// Mitsubishi GX Works2 project: ZhaoQing_HuaCheng1_12_5_12_52   PLC: Q03UDE

TYPE ConveyorIO : STRUCT
  xCWPresent : BOOL;  (* 正转检测有无传感器 *)
  xCCWPresent : BOOL;  (* 反转检测有无传感器 *)
  xLoad : BOOL;  (* 上料请求 *)
  xUnload : BOOL;  (* 下料请求 *)
  xMotorCW : BOOL;  (* 电机正转 *)
  xMotorCCW : BOOL;  (* 电机反转 *)
  xEmpty : BOOL;  (* 线体状态为空 *)
  xNextRun : BOOL;  (* 下段线体运行 *)
  xLastRun : BOOL;  (* 上段线体运行 *)
  xUnloadCCW : BOOL;  (* 下料为反转 *)
  xloadCCW : BOOL;  (* 上料为反转 *)
  xLeave : BOOL;  (* 已经离开 *)
  xAuto : BOOL;  (* 自动 *)
  xManual : BOOL;  (* 手动 *)
  xForward : BOOL;  (* 正转手动 *)
  xBackward : BOOL;  (* 反转手动 *)
  strProductSerial : STRING[4];  (* 产品信息 *)
  xEStop : BOOL;  (* 急停 *)
  xReset : BOOL;  (* 复位 *)
  iProductCategory : INT;  (* 产品类型0：无料1：正极  2：负极 3：隔膜 4：空料架 *)
  xBusy : BOOL;  (* 工作中 *)
  tLeaveDelay : TIME;  (* 离开延时设置 *)
  xPutInto : BOOL;  (* 线体直接投入物料 *)
  xLoadAlarrm : BOOL;  (* 上料报警 *)
  xUnloadAlarm : BOOL;  (* 下料报警 *)
END_STRUCT END_TYPE

TYPE ShuttleCarIO : STRUCT
  xAuto : BOOL;  (* 自动 *)
  xManual : BOOL;  (* 手动 *)
  xReady : BOOL;  (* 准备就绪 *)
  xForward : BOOL;  (* 正转 *)
  xBackward : BOOL;  (* 反转 *)
  diCurrentPos : DINT;  (* 当前位置 *)
  diDestinationPos : DINT;  (* 目标位置 *)
  xCW : BOOL;  (* 正转输出 *)
  xCCW : BOOL;  (* 反转输出 *)
  xBrake : BOOL;  (* 刹车 *)
  xHomeSwitch : BOOL;  (* 零位接近开关 *)
  xPosLimit : BOOL;  (* 正限位 *)
  xNegLimit : BOOL;  (* 负限位 *)
  xMDIExe : BOOL;  (* MDI开始 *)
  xMDIDone : BOOL;  (* MDI 完成 *)
  xPassLimit : BOOL;  (* 限位屏蔽 *)
  xPosLimitCatch : BOOL;  (* 正限位捕捉 *)
  xNegLimitCatch : BOOL;  (* 负限位捕捉 *)
  xHomeExe : BOOL;  (* 开始寻零 *)
  xHomeDone : BOOL;  (* 寻零完成 *)
  xHomeBusy : BOOL;  (* 寻零中 *)
  xHomeFailed : BOOL;  (* 寻零失败 *)
  xBusy : BOOL;  (* 工作中 *)
  xReset : BOOL;  (* 复位 *)
  xEStop : BOOL;  (* 急停 *)
END_STRUCT END_TYPE

TYPE SwitchIO : STRUCT
  xAuto : BOOL;
  xManual : BOOL;
  xEStop : BOOL;
  xReset : BOOL;
  xLiftCylinderRetractDetect : BOOL;
  xLiftCylinderExtendDetect : BOOL;
  xLiftCylinderRetract : BOOL;
  xLiftCylinderExtend : BOOL;
  xEntryBarCylinderRetract : BOOL;
  xLiftCylinderExtendInit : BOOL;
  xEntryEnable : BOOL;
  xExitEnable : BOOL;
  xExitBarCylinderRetract : BOOL;
  xSwithEnable : BOOL;
  xLiftCylinderRetractButton : BOOL;
  xLiftCylinderExtendButton : BOOL;
  xEntryBarCylinderRetractButton : BOOL;
  xExitBarCylinderRetractButton : BOOL;
END_STRUCT END_TYPE

// global labels: Global1
VAR_GLOBAL
  g_xAuto : BOOL;
  g_xManual : BOOL;
  g_xEStop AT X23 : BOOL;
  g_xReset AT X20 : BOOL;
  g_xStackLampRed AT Y120 : BOOL;
  g_xStackLampAmber AT Y121 : BOOL;
  g_xStackLampGreen AT Y122 : BOOL;
  g_xBuzzer AT Y123 : BOOL;
  g_xStop AT M2 : BOOL;
  g_xLocalAutoStart AT M1 : BOOL;
  g_xRemoteAutoStart AT M0 : BOOL;
  g_xRemoteAuto AT M10 : BOOL;
  g_iState AT D40 : INT;
  g_iLocalAutoStep : INT;
END_VAR

// task Task_01 (event TRUE, interval 0, priority 31): POU, Start, UDP

PROGRAM POU
VAR
  H3000Conveyor1 : Conveyor;
  H3000Conveyor1IO : ConveyorIO;
  H3000Conveyor2 : Conveyor;
  H3000Conveyor2IO : ConveyorIO;
  H3000Conveyor3 : Conveyor;
  H3000Conveyor3IO : ConveyorIO;
  H3000Conveyor4 : Conveyor;
  H3000Conveyor4IO : ConveyorIO;
  H3000Conveyor5 : Conveyor;
  H3000Conveyor5IO : ConveyorIO;
  H3000Conveyor6 : Conveyor;
  H3000Conveyor6IO : ConveyorIO;
  H3000Conveyor7 : Conveyor;
  H3000Conveyor7IO : ConveyorIO;
  H3000Conveyor8 : Conveyor;
  H3000Conveyor8IO : ConveyorIO;
  H3000Conveyor9 : Conveyor;
  H3000Conveyor9IO : ConveyorIO;
  H3000Conveyor10 : Conveyor;
  H3000Conveyor10IO : ConveyorIO;
  H3000ChemConveyor1 : Conveyor;
  H3000ChemConveyor1IO : ConveyorIO;
  H3000ChemConveyor2 : Conveyor;
  H3000ChemConveyor2IO : ConveyorIO;
  H3000ChemConveyor3 : Conveyor;
  H3000ChemConveyor3IO : ConveyorIO;
  Lifter1 : ShuttleCar;
  Lifter1IO : ShuttleCarIO;
  Conveyor1 : Conveyor;
  Conveyor1IO : ConveyorIO;
  Lifter2 : ShuttleCar;
  Lifter2IO : ShuttleCarIO;
  Conveyor2 : Conveyor;
  Conveyor2IO : ConveyorIO;
  H2200Conveyor1 : Conveyor;
  H2200Conveyor1IO : ConveyorIO;
  H2200Conveyor2 : Conveyor;
  H2200Conveyor2IO : ConveyorIO;
  H2200Conveyor3 : Conveyor;
  H2200Conveyor3IO : ConveyorIO;
  H2200Conveyor4 : Conveyor;
  H2200Conveyor4IO : ConveyorIO;
  H2200Conveyor5 : Conveyor;
  H2200Conveyor5IO : ConveyorIO;
  H2200Conveyor6 : Conveyor;
  H2200Conveyor6IO : ConveyorIO;
  H2200Conveyor7 : Conveyor;
  H2200Conveyor7IO : ConveyorIO;
  H2200Conveyor8 : Conveyor;
  H2200Conveyor8IO : ConveyorIO;
  H2200Conveyor9 : Conveyor;
  H2200Conveyor9IO : ConveyorIO;
  H2200Conveyor10 : Conveyor;
  H2200Conveyor10IO : ConveyorIO;
  H1000Conveyor1 : Conveyor;
  H1000Conveyor1IO : ConveyorIO;
  H1000Conveyor2 : Conveyor;
  H1000Conveyor2IO : ConveyorIO;
  H1000Conveyor3 : Conveyor;
  H1000Conveyor3IO : ConveyorIO;
  H1000Conveyor4 : Conveyor;
  H1000Conveyor4IO : ConveyorIO;
  H1000Conveyor5 : Conveyor;
  H1000Conveyor5IO : ConveyorIO;
  H1000Conveyor6 : Conveyor;
  H1000Conveyor6IO : ConveyorIO;
  H1000Conveyor7 : Conveyor;
  H1000Conveyor7IO : ConveyorIO;
  H1000Conveyor8 : Conveyor;
  H1000Conveyor8IO : ConveyorIO;
  H1000Conveyor9 : Conveyor;
  H1000Conveyor9IO : ConveyorIO;
  H3000SwitchQuadPackage : Switch;
  H3000SwitchQuadPackageIO : SwitchIO;
  H3000SwitchChem : Switch;
  H3000SwitchChemIO : SwitchIO;
  H3000SwitchPackageConveyorIn : ConveyorIO;
  H3000SwitchPackageConveyorOut : ConveyorIO;
  H850Switch : Switch;
  H850SwitchIO : SwitchIO;
  H850SwitchConveyorIn : ConveyorIO;
  H850SwitchConveyorOut : ConveyorIO;
  H850Conveyor8 : Conveyor;
  H850Conveyor8IO : ConveyorIO;
  H1000Conveyor10 : Conveyor;
  H1000Conveyor10IO : ConveyorIO;
  H3000SwitchChemConveyorIn : ConveyorIO;
  H3000SwitchChemConveyorOut : ConveyorIO;
END_VAR
H3000SwitchQuadPackage(ConveyorEntryIO:=H3000SwitchPackageConveyorIn ,
                                                        ConveyorExitIO:=H3000SwitchPackageConveyorOut ,
                                                        SwitchIO:=H3000SwitchQuadPackageIO );
H3000SwitchQuadPackageIO.xAuto:=g_xAuto;
H3000SwitchQuadPackageIO.xManual:=g_xManual;
H3000SwitchQuadPackageIO.xReset:=g_xReset;
H3000SwitchQuadPackageIO.xLiftCylinderExtendButton:=M75;
H3000SwitchQuadPackageIO.xLiftCylinderRetractButton:=M76;
H3000SwitchQuadPackageIO.xExitBarCylinderRetractButton:=M83;
Y128:=H3000SwitchQuadPackageIO.xEXITBarCylinderRetract;
Y12C:=H3000SwitchQuadPackageIO.xLiftCylinderExtend;
Y12A:=H3000SwitchQuadPackageIO.xLiftCylinderRetract;
H3000SwitchQuadPackageIO.xLiftCylinderExtendDetect:=X29;
H3000SwitchQuadPackageIO.xLiftCylinderRetractDetect:=X2A;
H3000SwitchPackageConveyorIn.xForward:=M77;
H3000SwitchPackageConveyorIn.xCWPresent:=X28;
Y187:=H3000SwitchPackageConveyorIn.xMotorCW;
H3000SwitchPackageConveyorOut.xForward:=M78;
H3000SwitchPackageConveyorOut.xCWPresent:=X2B;
Y12B:=H3000SwitchPackageConveyorOut.xMotorCW;

H3000SwitchChem(ConveyorEntryIO:=H3000SwitchChemConveyorIn ,
                                                        ConveyorExitIO:=H3000SwitchChemConveyorOut ,
                                                        SwitchIO:=H3000SwitchChemIO );
H3000SwitchChemIO.xAuto:=g_xAuto;
H3000SwitchChemIO.xManual:=g_xManual;
H3000SwitchChemIO.xReset:=g_xReset;
H3000SwitchChemIO.xLiftCylinderExtendButton:=M79;
H3000SwitchChemIO.xLiftCylinderRetractButton:=M80;
Y129:=H3000SwitchChemIO.xLiftCylinderExtend;
Y12D:=H3000SwitchChemIO.xLiftCylinderRetract;
H3000SwitchChemIO.xLiftCylinderExtendDetect:=X2C;
H3000SwitchChemIO.xLiftCylinderRetractDetect:=X2D;
H3000SwitchChemConveyorIn.xForward:=M81;
H3000SwitchChemConveyorIn.xCWPresent:=X2E;
(*Y19B:=H3000SwitchPackageConveyorIn.xMotorCW;*)
H3000SwitchChemConveyorOut.xForward:=M82;
H3000SwitchChemConveyorOut.xCWPresent:=X2E;
Y12E:=H3000SwitchChemConveyorOut.xMotorCW;
H3000SwitchChemIO.xSwithEnable:=1;

Lifter1(ShuttleCarInOut:=Lifter1IO);
ShuttleCarCurrentPosition( X8C OR X8D ,X8C ,X8D, FALSE, Lifter1IO.diCurrentPos );
Lifter1IO.xAuto:=g_xAuto;
Lifter1IO.xManual:=g_xManual;
Lifter1IO.xEStop:=g_xEStop;
Lifter1IO.xReset:=g_xReset;
Lifter1IO.xReady:=X24;
Lifter1Io.xForward:=M50 OR X91;
Lifter1IO.xBackward:=M51 OR X92;
Lifter1IO.xPosLimit:=X8E;
Lifter1IO.xNegLimit:=X8F;
Y18D:=Lifter1IO.xCW;
Y18E:=Lifter1IO.xCCW;
Y192:=Lifter1IO.xBrake;

Conveyor1(ConveyorMotor:=Conveyor1IO);
Conveyor1IO.xAuto:=g_xAuto;
Conveyor1IO.xManual:=g_xManual;
Conveyor1IO.xReset:=g_xReset;
Conveyor1IO.tLeaveDelay:=T#2s;
Conveyor1IO.xForward:=M52;
Conveyor1IO.xBackward:=M53;
Conveyor1IO.xCWPresent:=X193;
Conveyor1IO.xCCWPresent:=X194;
Y18B:=Conveyor1IO.xMotorCW;
Y18C:=Conveyor1IO.xMotorCCW;

Lifter2(ShuttleCarInOut:=Lifter2IO);
ShuttleCarCurrentPosition( X96 OR X97 ,X96 ,X97, FALSE, Lifter2IO.diCurrentPos );
Lifter2IO.xAuto:=g_xAuto;
Lifter2IO.xManual:=g_xManual;
Lifter2IO.xEStop:=g_xEStop;
Lifter2IO.xReset:=g_xReset;
Lifter2IO.xReady:=X25;
Lifter2Io.xForward:=M54 OR X9B;
Lifter2IO.xBackward:=M55 OR X9C;
Lifter2IO.xPosLimit:=X98;
Lifter2IO.xNegLimit:=X99;
Y193:=Lifter2IO.xCW;
Y194:=Lifter2IO.xCCW;
Y198:=Lifter2IO.xBrake;

Conveyor2(ConveyorMotor:=Conveyor2IO);
Conveyor2IO.xAuto:=g_xAuto;
Conveyor2IO.xManual:=g_xManual;
Conveyor2IO.xReset:=g_xReset;
Conveyor2IO.tLeaveDelay:=T#2s;
Conveyor2IO.xForward:=M56;
Conveyor2IO.xBackward:=M57;
Conveyor2IO.xCWPresent:=X93;
Conveyor2IO.xCCWPresent:=X94;
Y199:=Conveyor2IO.xMotorCW;
Y19A:=Conveyor2IO.xMotorCCW;


H3000Conveyor1(ConveyorMotor:=H3000Conveyor1IO);
H3000Conveyor1IO.xAuto:=g_xAuto;
H3000Conveyor1IO.xManual:=g_xManual;
H3000Conveyor1IO.xReset:=g_xReset;
H3000Conveyor1IO.tLeaveDelay:=t#2s;
H3000Conveyor1IO.xForward:=M30;
H3000Conveyor1IO.xCWPresent:=X2F;
Y12F:=H3000Conveyor1IO.xMotorCW;

H3000Conveyor2(ConveyorMotor:=H3000Conveyor2IO);
H3000Conveyor2IO.xAuto:=g_xAuto;
H3000Conveyor2IO.xManual:=g_xManual;
H3000Conveyor2IO.xReset:=g_xReset;
H3000Conveyor2IO.tLeaveDelay:=t#2s;
H3000Conveyor2IO.xForward:=M31;
H3000Conveyor2IO.xCWPresent:=X30;
Y130:=H3000Conveyor2IO.xMotorCW;

H3000Conveyor3(ConveyorMotor:=H3000Conveyor3IO);
H3000Conveyor3IO.xAuto:=g_xAuto;
H3000Conveyor3IO.xManual:=g_xManual;
H3000Conveyor3IO.xReset:=g_xReset;
H3000Conveyor3IO.tLeaveDelay:=t#2s;
H3000Conveyor3IO.xForward:=M32;
H3000Conveyor3IO.xCWPresent:=X31;
Y131:=H3000Conveyor3IO.xMotorCW;

H3000Conveyor4(ConveyorMotor:=H3000Conveyor4IO);
H3000Conveyor4IO.xAuto:=g_xAuto;
H3000Conveyor4IO.xManual:=g_xManual;
H3000Conveyor4IO.xReset:=g_xReset;
H3000Conveyor4IO.tLeaveDelay:=t#2s;
H3000Conveyor4IO.xForward:=M33;
H3000Conveyor4IO.xCWPresent:=X32;
Y132:=H3000Conveyor4IO.xMotorCW;

H3000Conveyor5(ConveyorMotor:=H3000Conveyor5IO);
H3000Conveyor5IO.xAuto:=g_xAuto;
H3000Conveyor5IO.xManual:=g_xManual;
H3000Conveyor5IO.xReset:=g_xReset;
H3000Conveyor5IO.tLeaveDelay:=t#2s;
H3000Conveyor5IO.xForward:=M34;
H3000Conveyor5IO.xCWPresent:=X33;
Y133:=H3000Conveyor5IO.xMotorCW;

H3000Conveyor6(ConveyorMotor:=H3000Conveyor6IO);
H3000Conveyor6IO.xAuto:=g_xAuto;
H3000Conveyor6IO.xManual:=g_xManual;
H3000Conveyor6IO.xReset:=g_xReset;
H3000Conveyor6IO.tLeaveDelay:=t#2s;
H3000Conveyor6IO.xForward:=M34;
H3000Conveyor6IO.xCWPresent:=X34;
Y134:=H3000Conveyor6IO.xMotorCW;

H3000Conveyor7(ConveyorMotor:=H3000Conveyor7IO);
H3000Conveyor7IO.xAuto:=g_xAuto;
H3000Conveyor7IO.xManual:=g_xManual;
H3000Conveyor7IO.xReset:=g_xReset;
H3000Conveyor7IO.tLeaveDelay:=t#2s;
H3000Conveyor7IO.xForward:=M35;
H3000Conveyor7IO.xCWPresent:=X35;
Y135:=H3000Conveyor7IO.xMotorCW;

H3000Conveyor8(ConveyorMotor:=H3000Conveyor8IO);
H3000Conveyor8IO.xAuto:=g_xAuto;
H3000Conveyor8IO.xManual:=g_xManual;
H3000Conveyor8IO.xReset:=g_xReset;
H3000Conveyor8IO.tLeaveDelay:=t#2s;
H3000Conveyor8IO.xForward:=M36;
H3000Conveyor8IO.xCWPresent:=X36;
Y136:=H3000Conveyor8IO.xMotorCW;

H3000Conveyor9(ConveyorMotor:=H3000Conveyor9IO);
H3000Conveyor9IO.xAuto:=g_xAuto;
H3000Conveyor9IO.xManual:=g_xManual;
H3000Conveyor9IO.xReset:=g_xReset;
H3000Conveyor9IO.tLeaveDelay:=t#2s;
H3000Conveyor9IO.xForward:=M37;
H3000Conveyor9IO.xCWPresent:=X37;
Y137:=H3000Conveyor9IO.xMotorCW;

H3000Conveyor10(ConveyorMotor:=H3000Conveyor10IO);
H3000Conveyor10IO.xAuto:=g_xAuto;
H3000Conveyor10IO.xManual:=g_xManual;
H3000Conveyor10IO.xReset:=g_xReset;
H3000Conveyor10IO.tLeaveDelay:=t#2s;
H3000Conveyor10IO.xForward:=M38;
H3000Conveyor10IO.xCWPresent:=X38;
Y138:=H3000Conveyor10IO.xMotorCW;

H3000ChemConveyor1(ConveyorMotor:=H3000ChemConveyor1IO);
H3000ChemConveyor1IO.xAuto:=g_xAuto;
H3000ChemConveyor1IO.xManual:=g_xManual;
H3000ChemConveyor1IO.xReset:=g_xReset;
H3000ChemConveyor1IO.tLeaveDelay:=t#2s;
H3000ChemConveyor1IO.xForward:=M39;
H3000ChemConveyor1IO.xCWPresent:=X39;
Y139:=H3000ChemConveyor1IO.xMotorCW;

H3000ChemConveyor2(ConveyorMotor:=H3000ChemConveyor2IO);
H3000ChemConveyor2IO.xAuto:=g_xAuto;
H3000ChemConveyor2IO.xManual:=g_xManual;
H3000ChemConveyor2IO.xReset:=g_xReset;
H3000ChemConveyor2IO.tLeaveDelay:=t#2s;
H3000ChemConveyor2IO.xForward:=M40;
H3000ChemConveyor2IO.xCWPresent:=X3A;
Y13A:=H3000ChemConveyor2IO.xMotorCW;

H3000ChemConveyor3(ConveyorMotor:=H3000ChemConveyor3IO);
H3000ChemConveyor3IO.xAuto:=g_xAuto;
H3000ChemConveyor3IO.xManual:=g_xManual;
H3000ChemConveyor3IO.xReset:=g_xReset;
H3000ChemConveyor3IO.tLeaveDelay:=t#2s;
H3000ChemConveyor3IO.xForward:=M41;
H3000ChemConveyor3IO.xCWPresent:=X3B;
Y13B:=H3000ChemConveyor3IO.xMotorCW;

H2200Conveyor1(ConveyorMotor:=H2200Conveyor1IO);
H2200Conveyor1IO.xAuto:=g_xAuto;
H2200Conveyor1IO.xManual:=g_xManual;
H2200Conveyor1IO.xReset:=g_xReset;
H2200Conveyor1IO.tLeaveDelay:=t#2s;
H2200Conveyor1IO.xForward:=M42;
H2200Conveyor1IO.xCWPresent:=X3F;
Y13F:=H2200Conveyor1IO.xMotorCW;

H2200Conveyor2(ConveyorMotor:=H2200Conveyor2IO);
H2200Conveyor2IO.xAuto:=g_xAuto;
H2200Conveyor2IO.xManual:=g_xManual;
H2200Conveyor2IO.xReset:=g_xReset;
H2200Conveyor2IO.tLeaveDelay:=t#2s;
H2200Conveyor2IO.xForward:=M43;
H2200Conveyor2IO.xCWPresent:=X40;
Y140:=H2200Conveyor2IO.xMotorCW;

H2200Conveyor3(ConveyorMotor:=H2200Conveyor3IO);
H2200Conveyor3IO.xAuto:=g_xAuto;
H2200Conveyor3IO.xManual:=g_xManual;
H2200Conveyor3IO.xReset:=g_xReset;
H2200Conveyor3IO.tLeaveDelay:=t#2s;
H2200Conveyor3IO.xForward:=M44;
H2200Conveyor3IO.xCWPresent:=X41;
Y141:=H2200Conveyor2IO.xMotorCW;

H2200Conveyor4(ConveyorMotor:=H2200Conveyor4IO);
H2200Conveyor4IO.xAuto:=g_xAuto;
H2200Conveyor4IO.xManual:=g_xManual;
H2200Conveyor4IO.xReset:=g_xReset;
H2200Conveyor4IO.tLeaveDelay:=t#2s;
H2200Conveyor4IO.xForward:=M45;
H2200Conveyor4IO.xCWPresent:=X42;
Y142:=H2200Conveyor2IO.xMotorCW;

H2200Conveyor5(ConveyorMotor:=H2200Conveyor5IO);
H2200Conveyor5IO.xAuto:=g_xAuto;
H2200Conveyor5IO.xManual:=g_xManual;
H2200Conveyor5IO.xReset:=g_xReset;
H2200Conveyor5IO.tLeaveDelay:=t#2s;
H2200Conveyor5IO.xForward:=M46;
H2200Conveyor5IO.xCWPresent:=X43;
Y143:=H2200Conveyor2IO.xMotorCW;

H2200Conveyor6(ConveyorMotor:=H2200Conveyor6IO);
H2200Conveyor6IO.xAuto:=g_xAuto;
H2200Conveyor6IO.xManual:=g_xManual;
H2200Conveyor6IO.xReset:=g_xReset;
H2200Conveyor6IO.tLeaveDelay:=t#2s;
H2200Conveyor6IO.xForward:=M47;
H2200Conveyor6IO.xCWPresent:=X44;
Y144:=H2200Conveyor6IO.xMotorCW;

H2200Conveyor7(ConveyorMotor:=H2200Conveyor7IO);
H2200Conveyor7IO.xAuto:=g_xAuto;
H2200Conveyor7IO.xManual:=g_xManual;
H2200Conveyor7IO.xReset:=g_xReset;
H2200Conveyor7IO.tLeaveDelay:=t#2s;
H2200Conveyor7IO.xForward:=M48;
H2200Conveyor7IO.xCWPresent:=X45;
Y145:=H2200Conveyor7IO.xMotorCW;

H2200Conveyor8(ConveyorMotor:=H2200Conveyor8IO);
H2200Conveyor8IO.xAuto:=g_xAuto;
H2200Conveyor8IO.xManual:=g_xManual;
H2200Conveyor8IO.xReset:=g_xReset;
H2200Conveyor8IO.tLeaveDelay:=t#2s;
H2200Conveyor8IO.xForward:=M49;
H2200Conveyor8IO.xCWPresent:=X46;
Y146:=H2200Conveyor8IO.xMotorCW;

H2200Conveyor9(ConveyorMotor:=H2200Conveyor9IO);
H2200Conveyor9IO.xAuto:=g_xAuto;
H2200Conveyor9IO.xManual:=g_xManual;
H2200Conveyor9IO.xReset:=g_xReset;
H2200Conveyor9IO.tLeaveDelay:=t#2s;
H2200Conveyor9IO.xForward:=M58;
H2200Conveyor9IO.xCWPresent:=X47;
Y147:=H2200Conveyor9IO.xMotorCW;

H2200Conveyor10(ConveyorMotor:=H2200Conveyor10IO);
H2200Conveyor10IO.xAuto:=g_xAuto;
H2200Conveyor10IO.xManual:=g_xManual;
H2200Conveyor10IO.xReset:=g_xReset;
H2200Conveyor10IO.tLeaveDelay:=t#2s;
H2200Conveyor10IO.xForward:=M59;
H2200Conveyor10IO.xCWPresent:=X48;
Y148:=H2200Conveyor10IO.xMotorCW;

H1000Conveyor1(ConveyorMotor:=H1000Conveyor1IO);
H1000Conveyor1IO.xAuto:=g_xAuto;
H1000Conveyor1IO.xManual:=g_xManual;
H1000Conveyor1IO.xReset:=g_xReset;
H1000Conveyor1IO.tLeaveDelay:=t#2s;
H1000Conveyor1IO.xForward:=M60;
H1000Conveyor1IO.xCWPresent:=X49;
Y149:=H1000Conveyor1IO.xMotorCW;

H1000Conveyor2(ConveyorMotor:=H1000Conveyor2IO);
H1000Conveyor2IO.xAuto:=g_xAuto;
H1000Conveyor2IO.xManual:=g_xManual;
H1000Conveyor2IO.xReset:=g_xReset;
H1000Conveyor2IO.tLeaveDelay:=t#2s;
H1000Conveyor2IO.xForward:=M61;
H1000Conveyor2IO.xCWPresent:=X4A;
Y14A:=H1000Conveyor2IO.xMotorCW;

H1000Conveyor3(ConveyorMotor:=H1000Conveyor3IO);
H1000Conveyor3IO.xAuto:=g_xAuto;
H1000Conveyor3IO.xManual:=g_xManual;
H1000Conveyor3IO.xReset:=g_xReset;
H1000Conveyor3IO.tLeaveDelay:=t#2s;
H1000Conveyor3IO.xForward:=M62;
H1000Conveyor3IO.xCWPresent:=X4B;
Y14B:=H1000Conveyor3IO.xMotorCW;

H1000Conveyor4(ConveyorMotor:=H1000Conveyor4IO);
H1000Conveyor4IO.xAuto:=g_xAuto;
H1000Conveyor4IO.xManual:=g_xManual;
H1000Conveyor4IO.xReset:=g_xReset;
H1000Conveyor4IO.tLeaveDelay:=t#2s;
H1000Conveyor4IO.xForward:=M63;
H1000Conveyor4IO.xCWPresent:=X4C;
Y14C:=H1000Conveyor4IO.xMotorCW;

H1000Conveyor5(ConveyorMotor:=H1000Conveyor5IO);
H1000Conveyor5IO.xAuto:=g_xAuto;
H1000Conveyor5IO.xManual:=g_xManual;
H1000Conveyor5IO.xReset:=g_xReset;
H1000Conveyor5IO.tLeaveDelay:=t#2s;
H1000Conveyor5IO.xForward:=M64;
H1000Conveyor5IO.xCWPresent:=X4D;
Y14D:=H1000Conveyor1IO.xMotorCW;

H1000Conveyor6(ConveyorMotor:=H1000Conveyor6IO);
H1000Conveyor6IO.xAuto:=g_xAuto;
H1000Conveyor6IO.xManual:=g_xManual;
H1000Conveyor6IO.xReset:=g_xReset;
H1000Conveyor6IO.tLeaveDelay:=t#2s;
H1000Conveyor6IO.xForward:=M65;
H1000Conveyor6IO.xCWPresent:=X4E;
Y14E:=H1000Conveyor1IO.xMotorCW;

H1000Conveyor7(ConveyorMotor:=H1000Conveyor7IO);
H1000Conveyor7IO.xAuto:=g_xAuto;
H1000Conveyor7IO.xManual:=g_xManual;
H1000Conveyor7IO.xReset:=g_xReset;
H1000Conveyor7IO.tLeaveDelay:=t#2s;
H1000Conveyor7IO.xForward:=M66;
H1000Conveyor7IO.xCWPresent:=X4F;
Y14F:=H1000Conveyor1IO.xMotorCW;

H1000Conveyor8(ConveyorMotor:=H1000Conveyor8IO);
H1000Conveyor8IO.xAuto:=g_xAuto;
H1000Conveyor8IO.xManual:=g_xManual;
H1000Conveyor8IO.xReset:=g_xReset;
H1000Conveyor8IO.tLeaveDelay:=t#2s;
H1000Conveyor8IO.xForward:=M67;
H1000Conveyor8IO.xCWPresent:=X50;
Y150:=H1000Conveyor8IO.xMotorCW;

H850Switch(ConveyorEntryIO:=H850SwitchConveyorIn,ConveyorExitIO:=H850SwitchConveyorOut,SwitchIO:=H850SwitchIO);
H850SwitchIO.xAuto:=g_xAuto;
H850SwitchIO.xManual:=g_xManual;
H850SwitchIO.xReset:=g_xReset;
H850SwitchIO.xLiftCylinderExtendButton:=M71;
H850SwitchIO.xLiftCylinderRetractButton:=M72;
Y189:=H850SwitchIO.xLiftCylinderExtend;
Y188:=H850SwitchIO.xLiftCylinderRetract;
H850SwitchIO.xLiftCylinderExtendDetect:=X88;
H850SwitchIO.xLiftCylinderRetractDetect:=X89;
H850SwitchConveyorIn.xForward:=M70;
H850SwitchConveyorIn.xCWPresent:=XB4;
Y19B:=H850SwitchConveyorIn.xMotorCW;
H850SwitchConveyorOut.xForward:=M73;
H850SwitchConveyorOut.xCWPresent:=X8A;
Y18A:=H850SwitchConveyorOut.xMotorCW;


H850Conveyor8(ConveyorMotor:=H850Conveyor8IO);
H850Conveyor8IO.xAuto:=g_xAuto;
H850Conveyor8IO.xManual:=g_xManual;
H850Conveyor8IO.xReset:=g_xReset;
H850Conveyor8IO.tLeaveDelay:=t#2s;
H850Conveyor8IO.xForward:=M74;
H850Conveyor8IO.xCWPresent:=X7F;
Y17F:=H850Conveyor8IO.xMotorCW;

IF g_xAuto THEN
	H3000SwitchQuadPackageIO.xEntryEnable:=M881;
	H3000SwitchQuadPackageIO.xSwithEnable:=1;
	H3000SwitchQuadPackageio.xExitEnable:=H3000Conveyor1IO.xEmpty;
	H3000Conveyor1Io.xLoad:=H3000SwitchPackageConveyorOut.xNextRun;
	H3000Conveyor1IO.xUnload:=H3000Conveyor2IO.xEmpty;
	H3000Conveyor2IO.xLoad:=H3000Conveyor1IO.xNextRun;
	H3000Conveyor2IO.xUnload:=H3000Conveyor3IO.xEmpty;
	H3000Conveyor3IO.xLoad:=H3000Conveyor2IO.xNextRun;	
	H3000Conveyor3IO.xUnload:=H3000Conveyor4IO.xEmpty;
	H3000Conveyor4IO.xLoad:=H3000Conveyor3IO.xNextRun;
	H3000Conveyor4IO.xUnload:=H3000Conveyor5IO.xEmpty;
	H3000Conveyor5IO.xLoad:=H3000Conveyor4IO.xNextRun;
	H3000Conveyor5IO.xUnload:=H3000Conveyor6IO.xEmpty;
	H3000Conveyor6IO.xLoad:=H3000Conveyor5IO.xNextRun;
	H3000Conveyor6IO.xUnload:=H3000Conveyor7IO.xEmpty;
	H3000Conveyor7IO.xLoad:=H3000Conveyor6IO.xNextRun;
	H3000Conveyor7IO.xUnload:=H3000Conveyor8IO.xEmpty;
	H3000Conveyor8IO.xLoad:=H3000Conveyor7IO.xNextRun;	
	H3000Conveyor8IO.xUnload:=H3000Conveyor9IO.xEmpty;
	H3000Conveyor9IO.xLoad:=H3000Conveyor8IO.xNextRun;	
	H3000Conveyor9IO.xUnload:=H3000Conveyor10IO.xEmpty;
	H3000Conveyor10IO.xLoad:=H3000Conveyor9IO.xNextRun;
	
	H2200Conveyor1IO.xLoad:=M201;
	H2200Conveyor1IO.xUnload:=H2200Conveyor2IO.xEmpty;
	H2200Conveyor2IO.xLoad:=H2200Conveyor1IO.xNextRun;
	H2200Conveyor2IO.xUnload:=H2200Conveyor3IO.xEmpty;
	H2200Conveyor3IO.xLoad:=H2200Conveyor2IO.xNextRun;	
	H2200Conveyor3IO.xUnload:=H2200Conveyor4IO.xEmpty;
	H2200Conveyor4IO.xLoad:=H2200Conveyor3IO.xNextRun;
	H2200Conveyor4IO.xUnload:=H2200Conveyor5IO.xEmpty;
	H2200Conveyor5IO.xLoad:=H2200Conveyor4IO.xNextRun;
	H2200Conveyor5IO.xUnload:=H2200Conveyor6IO.xEmpty;
	H2200Conveyor6IO.xLoad:=H2200Conveyor5IO.xNextRun;
	H2200Conveyor6IO.xUnload:=H2200Conveyor7IO.xEmpty;
	H2200Conveyor7IO.xLoad:=H2200Conveyor6IO.xNextRun;
	H2200Conveyor7IO.xUnload:=H2200Conveyor8IO.xEmpty;
	H2200Conveyor8IO.xLoad:=H2200Conveyor7IO.xNextRun;	
	H2200Conveyor8IO.xUnload:=H2200Conveyor9IO.xEmpty;
	H2200Conveyor9IO.xLoad:=H2200Conveyor8IO.xNextRun;	
	H2200Conveyor9IO.xUnload:=H2200Conveyor10IO.xEmpty;
	H2200Conveyor10IO.xLoad:=H2200Conveyor9IO.xNextRun;
	
	H1000Conveyor10IO.xLoad:=M202;
	H1000Conveyor10IO.xUnload:=H1000Conveyor9IO.xEmpty;
    H1000Conveyor9IO.xLoad:=H1000Conveyor10IO.xNextRun;
    H1000Conveyor9IO.xUnload:=H1000Conveyor8IO.xEmpty;
    H1000Conveyor8IO.xLoad:=H1000Conveyor9IO.xNextRun;
    H1000Conveyor8IO.xUnload:=H1000Conveyor7IO.xEmpty;
    H1000Conveyor7IO.xLoad:=H1000Conveyor8IO.xNextRun;
    H1000Conveyor7IO.xUnload:=H1000Conveyor6IO.xEmpty;
    H1000Conveyor6IO.xLoad:=H1000Conveyor7IO.xNextRun;
    H1000Conveyor6IO.xUnload:=H1000Conveyor5IO.xEmpty;
    H1000Conveyor5IO.xLoad:=H1000Conveyor6IO.xNextRun;
    H1000Conveyor5IO.xUnload:=H1000Conveyor4IO.xEmpty;
    H1000Conveyor4IO.xLoad:=H1000Conveyor5IO.xNextRun;
    H1000Conveyor4IO.xUnload:=H1000Conveyor3IO.xEmpty;
    H1000Conveyor3IO.xLoad:=H1000Conveyor4IO.xNextRun;
    H1000Conveyor3IO.xUnload:=H1000Conveyor2IO.xEmpty;
    H1000Conveyor2IO.xLoad:=H1000Conveyor3IO.xNextRun;  
    H1000Conveyor2IO.xUnload:=H1000Conveyor1IO.xEmpty;
    H1000Conveyor1IO.xLoad:=H1000Conveyor2IO.xNextRun;      
	
	H850SwitchIO.xEntryEnable:=M880;
	H850SwitchIO.xSwithEnable:=1;
	H850SwitchIO.xExitEnable:=H850Conveyor8IO.xEmpty;
    H850Conveyor8IO.xLoad:=H850SwitchConveyorOut.xNextRun;
    
    
    
END_IF;
END_PROGRAM

FUNCTION_BLOCK Conveyor
VAR
  tRundelay : TIME;  (* 离开延时 *)
END_VAR
VAR_IN_OUT
  ConveyorMotor : ConveyorIO;  (* 输送线输入输出 *)
END_VAR
VAR
  iStep : INT;  (* 上料步骤 *)
  m_tLoadTimer : TIME;  (* 上料计时器 *)
  m_tUnloadTimer : TIME;  (* 下料计时器 *)
  m_tonLeaveDelay : TON;  (* 离开延时定时器 *)
  m_xLeaveDelayOut : BOOL;  (* 离开延时 *)
  m_tLeaveCurrentTime : TIME;
  m_tonLoadAlarm : TON;  (* 上料延时报警 *)
END_VAR
VAR CONSTANT
  LOAD_UNLOAD_TIME : TIME := T#30s;  (* 延时报警常量 *)
END_VAR
VAR
  m_tonUnloadAlam : TON;  (* 下料报警定时器 *)
END_VAR
(*////////////////////////////////////////////////////////////////////////////////////////////////////////////
//传输线控制FB块，可控制单方向线体，双向旋转线体，支持双向上下料            
//线体初始化后为空的情况下输入xLoad信号即可进行上料动作，使用xLoadCCW信号可反方向上料
//增加了产品信息和产品种类的储存，当传输线为空和上料进行标志位为零的情况下清除产品信息和产品种类
//使用方式是在置位xLoad信号后，把产品信息和产品种类传入，等下料后自动清零
//线体不为空的情况下使用xUnload信号可进行下料动作，物料有无传感器的下降沿后出发计时器，延时断开传输线旋转
//单方向传输线体把xLoadCCW、xUnloadCCW设置为零，双向线体上料方向和下料反向的,方向固定的 把xUnloadCCW设置为1
//双方向线体双向都能上下料的要根据上料的方向来设置xLoadCCW,xUnloadCCW
//增加工作中信号xBusy当电机正转 显示为工作中
//增加上下料超时报警，xLoadAlarm，xUnloadAlarm，设定时间在LOAD_UNLOAD_TIME常量上，现在设置的为30秒
//增加xPutInto信号，用于直接投入的物料，检测开关感应到后，直接进入下料流程，上升沿有效
//离开延时改为变量 iLeaveDelay 默认为0 离开检测开关离输送线尾端比较远的线体需要根据情况设定100ms为单位
//修改信息  修改后请增加版本
//YAO      V1.0
///////////////////////////////////////////////////////////////////////////////////////////////////////////
********************************************************)


IF ConveyorMotor.xAuto THEN
CASE iStep OF
	0:
	ConveyorMotor.xMotorCW:=0;
	ConveyorMotor.xMotorCCW:=0;
	ConveyorMotor.xNextRun:=0;

	IF (ConveyorMotor.xCWPresent OR ConveyorMotor.xCCWPresent) 
		AND ConveyorMotor.xEStop=0 
		AND ConveyorMotor.xLoadAlarrm = 0
		AND ConveyorMotor.xUnloadAlarm = 0 THEN
		iStep:=3;
		ConveyorMotor.xEmpty:=0;
		ELSE
		iStep:=1;
		ConveyorMotor.xEmpty:=1;
	END_IF;
		
	1: 
	IF ConveyorMotor.xLoad    
		AND ConveyorMotor.xMotorCW=0   
		AND ConveyorMotor.xMotorCCW=0   
		AND ConveyorMotor.xEmpty THEN	
		iStep:=2;
	END_IF;
	2: 
	IF ConveyorMotor.xloadCCW THEN
		ConveyorMotor.xMotorCCW:=1; 
		ConveyorMotor.xMotorCW:=0;
		IF ConveyorMotor.xCCWPresent THEN
			iStep:=3;
		END_IF;
		ELSE
	    ConveyorMotor.xMotorCW:=1;  
		ConveyorMotor.xMotorCCW:=0;
	    IF ConveyorMotor.xCWPresent THEN 	 
		    iStep:=3;
		END_IF;
	END_IF;
	3:
	ConveyorMotor.xMotorCW:=0;
	ConveyorMotor.xMotorCCW:=0;
	ConveyorMotor.xEmpty:=0;
	IF ConveyorMotor.xUnload THEN 
		iStep:=4;
	END_IF;
	4:	
	IF ConveyorMotor.xUnloadCCW THEN   
		ConveyorMotor.xMotorCCW:=1;  
		ConveyorMotor.xMotorCW:=0;

		ConveyorMotor.xLeave:=ldf(TRUE,ConveyorMotor.xCCWPresent) OR ConveyorMotor.xLeave;
		ELSE
	    ConveyorMotor.xMotorCW:=1;  
		ConveyorMotor.xMotorCCW:=0;
		ConveyorMotor.xLeave:=ldf(TRUE,ConveyorMotor.xCWPresent) OR ConveyorMotor.xLeave;
	END_IF;
	ConveyorMotor.xNextRun:=1; 
	m_tonLeaveDelay(IN:= ConveyorMotor.xLeave,PT:= ConveyorMotor.tLeaveDelay,Q:=m_xLeaveDelayOut ,ET:= m_tLeaveCurrentTime );	
	IF m_xLeaveDelayOut THEN
		ConveyorMotor.xMotorCW:=0;
		ConveyorMotor.xMotorCCW:=0;
		iStep:=0;
		ConveyorMotor.xNextRun:=0;
		ConveyorMotor.xLeave:=0;
		ConveyorMotor.xEmpty:=1;		
	END_IF;	
	IF NOT ConveyorMotor.xUnload THEN 
		istep:=0;
	END_IF;
END_CASE;
IF LDP(TRUE,ConveyorMotor.xPutInto) THEN
	iStep:=0;
END_IF;
END_IF;
IF ConveyorMotor.xEmpty AND NOT ConveyorMotor.xLoad THEN
	ConveyorMotor.strProductSerial:='';
	ConveyorMotor.iProductCategory:=0;
END_IF;
IF ConveyorMotor.xEStop OR ConveyorMotor.xReset THEN
	iStep:=0;
END_IF;	

IF ConveyorMotor.xManual THEN
	iStep:=0;

	IF ConveyorMotor.xForward 
		AND ConveyorMotor.xBackward=0 
		AND ConveyorMotor.xMotorCCW=0 THEN
		ConveyorMotor.xMotorCW:=1;
		ConveyorMotor.xMotorCCW:=0;
		ELSE
		ConveyorMotor.xMotorCW:=0;
	END_IF;

	IF ConveyorMotor.xBackward 
		AND ConveyorMotor.xForward=0 
		AND ConveyorMotor.xMotorCW=0  THEN
		ConveyorMotor.xMotorCCW:=1;
		conveyormotor.xMotorCW:=0;
		ELSE
		ConveyorMotor.xMotorCCW:=0;
	END_IF;
END_IF;
IF ConveyorMotor.xMotorCCW        
	OR ConveyorMotor.xMotorCW THEN  
	ConveyorMotor.xBusy:=1;
	ELSE
	ConveyorMotor.xBusy:=0;
END_IF;
m_tonLoadAlarm(IN:= iStep=2 ,PT:= LOAD_UNLOAD_TIME,Q:= ConveyorMotor.xLoadAlarrm ,ET:= m_tLoadTimer );
m_tonUnloadAlam(IN:= iStep=4,PT:= LOAD_UNLOAD_TIME,Q:= ConveyorMotor.xUnloadAlarm,ET:= m_tUnloadTimer );
(*OUT_T(iStep=2,m_tLoadTimer,LOAD_UNLOAD_TIME);
OUT_T(iStep=4,m_tUnloadTimer,LOAD_UNLOAD_TIME);
ConveyorMotor.xLoadAlarrm:=m_tLoadTimer.S;
ConveyorMotor.xUnloadAlarm:=m_tUnloadTimer.S;*)
END_FUNCTION_BLOCK

FUNCTION_BLOCK ShuttleCar
VAR_IN_OUT
  ShuttleCarInOut : ShuttleCarIO;
END_VAR
VAR
  m_xBrakeDelay : BOOL;  (* 刹车延时标志位 *)
  diCurrentPosRetain : DINT;
  m_tonBrakeDelay : TON;  (* 延时 *)
  m_tBrakeDelay : TIME;
  m_xBrake : BOOL;
  m_tBrakeDelayCurrentTime : TIME;
END_VAR
(*******************************************************************
输送小车程序，可用于使用认址片控制位置的输送车程序，可用于控制提升机，
使用了限位捕捉程序防止小车惯性过大冲过限位后继续行走，捕捉程序采用反
转复位，这样设计有弊端可能反转复位后车的位置并没有回到限位以内,当两个
限位同时碰到的时候，会使运料小车进入死锁状态，通过xPassLimit来解开死锁，
可以在触摸屏中使用一个带权限的按钮来进行控制，配合ShuttleCarCurrentPos
函数来计算位置信息
修改信息  修改后请增加版本
YAO      V1.0
********************************************************************)

ShuttleCarInOut.xPosLimitCatch:=LDF(TRUE,ShuttleCarInOut.xPosLimit) OR ShuttleCarInOut.xPosLimitCatch;
IF ShuttleCarInOut.xCCW THEN  
	ShuttleCarInOut.xPosLimitCatch:=0;
END_IF;

ShuttleCarInOut.xNegLimitCatch:=LDF(TRUE,ShuttleCarInOut.xNegLimit) OR ShuttleCarInOut.xNegLimitCatch;
IF ShuttleCarInOut.xCW THEN   
	ShuttleCarInOut.xNegLimitCatch:=0;  
END_IF;
IF ShuttleCarInOut.xPassLimit OR
	(ShuttleCarInOut.xNegLimitCatch 
	AND ShuttleCarInOut.xPosLimitCatch)  THEN  
	ShuttleCarInOut.xNegLimitCatch:=0; 
	ShuttleCarInOut.xPosLimitCatch:=0;
END_IF;

IF ShuttleCarInOut.xReady THEN	
    IF ShuttleCarInOut.xManual THEN  
	    IF ShuttleCarInOut.xForward 
			AND ShuttleCarInOut.xBackward=0 
			AND ShuttleCarInOut.xCCW=0 
			AND ShuttleCarInOut.xPosLimitCatch=0 
			AND ShuttleCarInOut.xEStop THEN
		    ShuttleCarInOut.xCW:=1;
		    ELSE
		    ShuttleCarInOut.xCW:=0;
	    END_IF;
	    IF ShuttleCarInOut.xBackward 
			AND ShuttleCarInOut.xForward=0 
			AND ShuttleCarInOut.xCW=0 
			AND ShuttleCarInOut.xNegLimitCatch=0 
			AND ShuttleCarInOut.xEStop THEN  
		    ShuttleCarInOut.xCCW:=1;
		    ELSE
		    ShuttleCarInOut.xCCW:=0;
	    END_IF;
    END_IF;
  IF ShuttleCarInOut.xAuto AND ShuttleCarInOut.xEStop THEN  
	  IF ShuttleCarInOut.xMDIExe AND ShuttleCarInOut.diDestinationPos<>0 THEN
	
	    IF ShuttleCarInOut.diCurrentPos<ShuttleCarInOut.diDestinationPos AND ShuttleCarInOut.xPosLimitCatch=0 THEN
			ShuttleCarInOut.xCW:=1;
			ShuttleCarInOut.xCCW:=0;
			ShuttleCarInOut.xMDIDone:=0;
		END_IF;

		IF ShuttleCarInOut.diCurrentPos>ShuttleCarInOut.diDestinationPos AND ShuttleCarInOut.xNegLimitCatch=0 THEN
			ShuttleCarInOut.xCCW:=1;
			ShuttleCarInOut.xCW:=0;
			ShuttleCarInOut.xMDIDone:=0;
		END_IF;
	
		IF ShuttleCarInOut.diCurrentPos=ShuttleCarInOut.diDestinationPos THEN
			ShuttleCarInOut.xCW:=0;
			ShuttleCarInOut.xCCW:=0;
			ShuttleCarInOut.xMDIDone:=1;
			ELSE
			ShuttleCarInOut.xMDIDone:=0;
		END_IF;

		IF ShuttleCarInOut.xPosLimitCatch THEN
			ShuttleCarInOut.xCW:=0;
			ShuttleCarInOut.xMDIDone:=0;
		END_IF;

		IF ShuttleCarInOut.xNegLimitCatch THEN
			ShuttleCarInOut.xCCW:=0;
			ShuttleCarInOut.xMDIDone:=0;
		END_IF;
		ELSE
		ShuttleCarInOut.xCW:=0;
		ShuttleCarInOut.xCCW:=0;
		ShuttleCarInOut.xMDIDone:=0;
	  END_IF;
	END_IF;
	ELSE
		ShuttleCarInOut.xCW:=0;
		ShuttleCarInOut.xCCW:=0;	
END_IF;

m_tonBrakeDelay(IN:=m_xBrakeDelay ,PT:= T#100ms,Q:=m_xBrake ,ET:= m_tBrakeDelayCurrentTime);
IF (ShuttleCarInOut.xCW OR ShuttleCarInOut.xCCW) AND ShuttleCarInOut.xReady=1 THEN
	ShuttleCarInOut.xBrake:=m_xBrake;
	m_xBrakeDelay:=1;
	ELSE
	ShuttleCarInOut.xBrake:=0;
	m_xBrakeDelay:=0;
END_IF;

IF ShuttleCarInOut.xEStop =0 THEN
	ShuttleCarInOut.xCW :=0;
	ShuttleCarInOut.xCCW:=0;
END_IF;

(*IF SM402 THEN 
	ShuttleCarInOut.diCurrentPos:=diCurrentPosRetain;
	ELSE
	diCurrentPosRetain:=ShuttleCarInOut.diCurrentPos;
END_IF;*)

IF ShuttleCarInOut.xCW OR ShuttleCarInOut.xCCW THEN
	ShuttleCarInOut.xBusy:=1;
	ELSE
	ShuttleCarInout.xBusy:=0;
END_IF;
END_FUNCTION_BLOCK

FUNCTION ShuttleCarCurrentPosition
VAR_INPUT
  xPosition1 : BOOL;
  xPosition2 : BOOL;
  xPosition3 : BOOL;
END_VAR
(************************************
计算输送车当前位置的函数
**************************************)
IF xPosition1 THEN
	ShuttleCarCurrentPosition:=1;
END_IF;
IF xPosition2 THEN
	ShuttleCarCurrentPosition:=2;
END_IF;
IF xPosition3 THEN
	ShuttleCarCurrentPosition:=3;
END_IF;
END_FUNCTION

FUNCTION_BLOCK Switch
VAR_IN_OUT
  ConveyorEntryIO : ConveyorIO;
END_VAR
VAR
  ConveyorEntry : Conveyor;
  m_tonEntryBarDelay : TON;  (* 进入阻挡器延时 *)
  m_tEntryBarDelay : TIME;
  m_xEntryBarDelay : BOOL;
END_VAR
VAR_IN_OUT
  ConveyorExitIO : ConveyorIO;
END_VAR
VAR
  m_tonLiftCylinderDelay : TON;  (* 顶升延时 *)
  m_xLiftCylinderDelay : BOOL;
  m_tLiftCylinderDelay : TIME;
  m_tonExitBarDelay : TON;  (* 退出阻挡器延时 *)
  m_tExitBarDelay : TIME;
  m_xExitBarDelay : BOOL;
END_VAR
VAR_IN_OUT
  SwitchIO : SwitchIO;
END_VAR
VAR
  iStep : INT;
  ConveyorExit : Conveyor;
END_VAR
ConveyorEntry(ConveyorMotor:=ConveyorEntryIO);
ConveyorEntryIO.xAuto:=SwitchIO.xAuto;
ConveyorEntryIO.xManual:=SwitchIO.xManual;
ConveyorEntryIO.xReset:=SwitchIO.xReset;
ConveyorEntryIO.tLeaveDelay:=T#2s;
ConveyorExit(ConveyorMotor:=ConveyorExitIO);
ConveyorExitIO.xAuto:=SwitchIO.xAuto;
ConveyorExitIO.xManual:=SwitchIO.xManual;
ConveyorExitIO.xReset:=SwitchIO.xReset;
ConveyorExitIO.tLeaveDelay:=T#5s;
IF SwitchIO.xAuto THEN
	CASE iStep OF
		0:(*初始化*)
		ConveyorEntryIO.xLoad:=0;
		ConveyorEntryIO.xUnload:=0;
		ConveyorEntryIO.xPutInto:=0;
		ConveyorExitIO.xLoad:=0;
		ConveyorExitIo.xUnload:=0;
		ConveyorExitIO.xPutInto:=0;
		SwitchIO.xEntryBarCylinderRetract:=0;
		SwitchIO.xExitBarCylinderRetract:=0;
		IF SwitchIO.xLiftCylinderExtendInit THEN
			SwitchIO.xLiftCylinderExtend:=1;
			SwitchIO.xLiftCylinderRetract:=0;
		    IF SwitchIO.xLiftCylinderExtendDetect THEN
			    iStep:=1;
		     END_IF; 
		ELSE
			SwitchIO.xLiftCylinderExtend:=0;
			SwitchIO.xLiftCylinderRetract:=1;	
		    IF SwitchIO.xLiftCylinderRetractDetect THEN
			    iStep:=1;
		    END_IF;		
		END_IF;
		1:(*上料*)
        IF SwitchIO.xEntryEnable THEN
        	SwitchIO.xEntryBarCylinderRetract:=1;
        	ConveyorEntryIO.xLoad:=1;
        END_IF;
        m_tonEntryBarDelay(IN:=SwitchIO.xEntryBarCylinderRetract ,PT:=T#1S ,Q:= m_xEntryBarDelay ,ET:= m_tEntryBarDelay );
        IF m_xEntryBarDelay THEN
        	ConveyorEntryIO.xPutInto:=1;
        END_IF;
        IF ConveyorEntryIO.xEmpty=0 THEN
        	SwitchIO.xEntryBarCylinderRetract:=0;
        	ConveyorEntryIO.xLoad:=0;
        	ConveyorExitIO.xPutInto:=1;
        END_IF;
        IF m_xLiftCylinderDelay AND  SwitchIO.xSwithEnable THEN
        	 iStep:=2;
        END_IF;
        IF SwitchIO.xSwithEnable=0 THEN
        	 iStep:=3;
        END_IF;
		2:(*顶升*)
			SwitchIO.xExitBarCylinderRetract:=0;
			ConveyorEntryIO.xPutInto:=0;(*复位进入初始化*)
		    IF SwitchIO.xLiftCylinderExtendInit THEN
			    SwitchIO.xLiftCylinderExtend:=0;
			    SwitchIO.xLiftCylinderRetract:=1;
		    ELSE
			    SwitchIO.xLiftCylinderExtend:=1;
			    SwitchIO.xLiftCylinderRetract:=0;			
		   END_IF;

		  IF SwitchIO.xLiftCylinderExtendInit THEN
		  	IF SwitchIO.xLiftCylinderRetractDetect THEN
		  		iStep:=4;
		  	END_IF;
		  	ELSE
		  	IF SwitchIO.xLiftCylinderExtendDetect THEN
		      iStep:=4; 
		  	END_IF;
		  END_IF;
		  3:(*放行*)	
		  	SwitchIO.xExitBarCylinderRetract:=1;
		  	iStep:=4;
		  4:(*下料*)
		  IF SwitchIO.xExitEnable  AND m_xExitBarDelay THEN		  
		  ConveyorExitIO.xUnload:=1;
		  END_IF;
		  IF ConveyorExitIO.xEmpty OR ConveyorEntryIO.xEmpty THEN
		  	COnveyorExitIO.xUnload:=0;
		  	ConveyorExitIO.xPutInto:=1;
		  	ConveyorEntryIO.xPutInto:=1;
			iStep:=0; 
		  END_IF;
	END_CASE;
        m_tonLiftCylinderDelay(IN:=NOT ConveyorEntryIO.xEmpty AND iStep=1 ,PT:= T#3S ,Q:= m_xLiftCylinderDelay ,ET:=m_tLiftCylinderDelay );
 		m_tonExitBarDelay(IN:=iStep=4 ,PT:= T#3s ,Q:= m_xExitBarDelay ,ET:= m_tExitBarDelay);
END_IF;
IF SwitchIO.xManual OR SwitchIO.xReset THEN
	iStep:=0;
	IF SwitchIO.xEntryBarCylinderRetractButton THEN
		SwitchIO.xEntryBarCylinderRetract:=1;
	ELSE
		SwitchIO.xEntryBarCylinderRetract:=0;
	END_IF;
		IF SwitchIO.xExitBarCylinderRetractButton THEN
		SwitchIO.xExitBarCylinderRetract:=1;
	ELSE
		SwitchIO.xExitBarCylinderRetract:=0;
		END_IF;
		IF SwitchIO.xLiftCylinderExtendButton AND NOT SwitchIO.xLiftCylinderRetractButton THEN
			SwitchIO.xLiftCylinderExtend:=1;
			SwitchIO.xLiftCylinderRetract:=0;
		END_IF;
		IF NOT SwitchIO.xLiftCylinderExtendButton AND  SwitchIO.xLiftCylinderRetractButton THEN
			SwitchIO.xLiftCylinderExtend:=0;
			SwitchIO.xLiftCylinderRetract:=1;
		END_IF;		
	END_IF;
END_FUNCTION_BLOCK

PROGRAM Start
IF g_xReset THEN
	SM50:=1;
ELSE
	SM50:=0;
END_IF;
CASE g_iState OF
	0: 
		g_xManual:=1;
		g_xAuto:=0;	
		g_xStackLampAmber:=1;
		g_xStackLampGreen:=0;
		g_xRemoteAuto:=0;
	1:
		g_xManual:=0;
		g_xAuto:=1;
		g_xStackLampGreen:=1;
		g_xStackLampAmber:=0;
		g_xRemoteAuto:=0;
	2:	
        g_xRemoteAuto:=1;
        g_xStackLampGreen:=1;
        g_xStackLampAmber:=0;
        g_xAuto:=0;
		g_xManual:=0;
END_CASE;
IF g_xLocalAutoStart THEN  
	g_iState:=1;
END_IF;

IF g_xStop OR g_xEStop=0 THEN 
	g_iState:=0;
END_IF;
IF g_xRemoteAutoStart THEN
	g_iState:=2;
END_IF;
END_PROGRAM

PROGRAM UDP
SP_SOCSND( SM413 , "U0" , K1 , D100, D200, M100 );
SP_SOCRCV( NOT M102 , "U0" , K1, D300 , D400 ,M102 );
END_PROGRAM
